// TIA Portal V15.1 export
DATA_BLOCK "PROAUTOMATOR_GLOBAL"   // DB10
// stored: AutoNumber true
   VAR
      ACTUATORS : Struct
         EV : Struct
            LimitSwitches : Struct
               Pippo : Bool;
               Work : Bool;
               Home : Bool;
            END_STRUCT;
            Conditions : Struct
               Home : Bool;
               Work : Bool;
            END_STRUCT;
            Commands : Struct
               Home : Bool;
               Work : Bool;
            END_STRUCT;
         END_STRUCT;
      END_STRUCT;
   END_VAR
BEGIN
END_DATA_BLOCK
